{attribute 'qualified_only'}
VAR_GLOBAL
	GrindingWheelMS:BOOL;
	GrindingWheelMS2:BOOL;
END_VAR

(* stored: Version 1.1.0.1, ProductVersion 3.1.4022.3
   GVL Grinder: Id {8db0d846-cda3-4d2f-b655-d2a023459888} *)
